(* IEC 61131-3 sources: plc-vscode/tests/st/all/trust-platform/conformance/cases/arithmetic/cfm_arithmetic_overflow_error_002, 1 file *)

(* ---- program.st ---- *)
PROGRAM Main
VAR
    a : INT := INT#32767;
    b : INT := INT#0;
END_VAR

b := a + INT#1;
END_PROGRAM
